{attribute 'GeneratedUsingTerminal: AT2041-0250-0021'}
{attribute addProperty BoxType "AT2041-0250-0021"}
{attribute addProperty Id "A_0101_AT2041_5250_0018_AT2041_5250AT2041_01D6DEDF80"}
{attribute addProperty CRC "949670676"}
{attribute addProperty Size "80"}
TYPE A_0043_AT2041_0250_0021_389AD314 EXTENDS AT2041_86175B41 :
STRUCT
	{attribute addProperty Name "A_0101_AT2041_5250_0018_AT2041_5250"}
	{attribute addProperty PreviousPort "A_0043(AT2041-0250-0021) : B"}
	A_0101_AT2041_5250_0018_AT2041_5250 : AT2041_01D6DEDF;
END_STRUCT
END_TYPE

(* stored: Version 1.2.0.0, ProductVersion 3.1.4024.9
   DUT A_0043_AT2041_0250_0021_389AD314: Id {125000a1-b302-4fc3-b383-4127cdae5a66} *)
